// TIA Portal V18 export
DATA_BLOCK "L1_Corr_plotter"   // DB42
{ S7_Optimized_Access := 'TRUE' }
VERSION : 0.1
// stored: AutoNumber true, DBAccessibleFromOPCUA true, DBAccessibleFromWebserver true, IsOnlyStoredInLoadMemory false, IsRetainMemResEnabled false, IsWriteProtectedInAS false, MemoryReserve 100
   VAR RETAIN
      "name" : WString[30];
      ID : DInt;
      corr_Y : Array[1..32] of LReal;
   END_VAR
BEGIN
END_DATA_BLOCK
